TYPE DUT_SERVER_STATEVALUEARRAY :
STRUCT
	StateValue0: DUT_STATEVALUES;
	StateValue1: DUT_STATEVALUES;
	StateValue2: DUT_STATEVALUES;
	StateValue3: DUT_STATEVALUES;
	StateValue4: DUT_STATEVALUES;
	StateValue5: DUT_STATEVALUES;
	StateValue6: DUT_STATEVALUES;
	StateValue7: DUT_STATEVALUES;
	StateValue8: DUT_STATEVALUES;
	StateValue9: DUT_STATEVALUES;
	StateValue10: DUT_STATEVALUES;
END_STRUCT
END_TYPE

(* stored: Version 1.1.0.1, ProductVersion 3.1.0.25
   DUT DUT_SERVER_STATEVALUEARRAY: Id {937403cb-800d-4270-af39-00ec252615ec} *)
